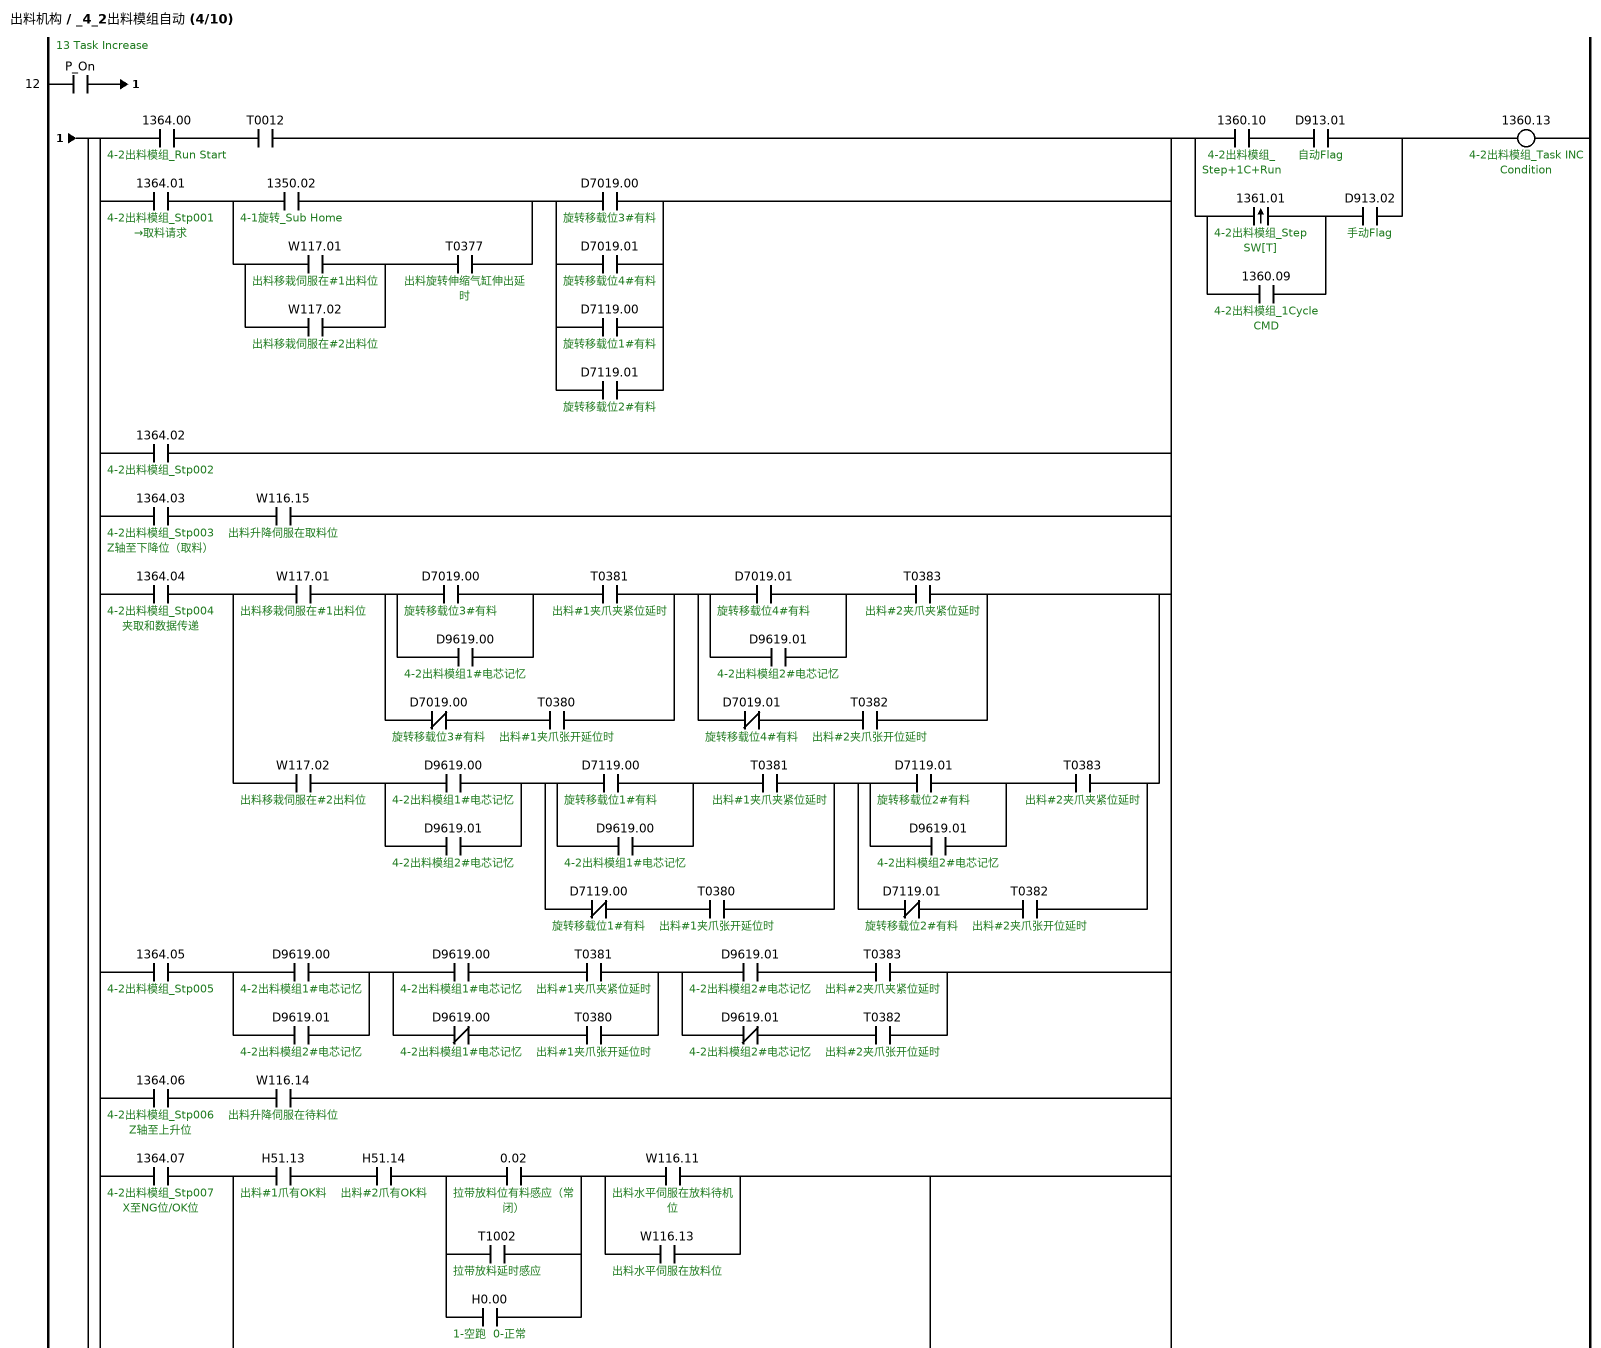
; [picture p384: 出料机构 / _4_2出料模组自动, rungs 12-12]

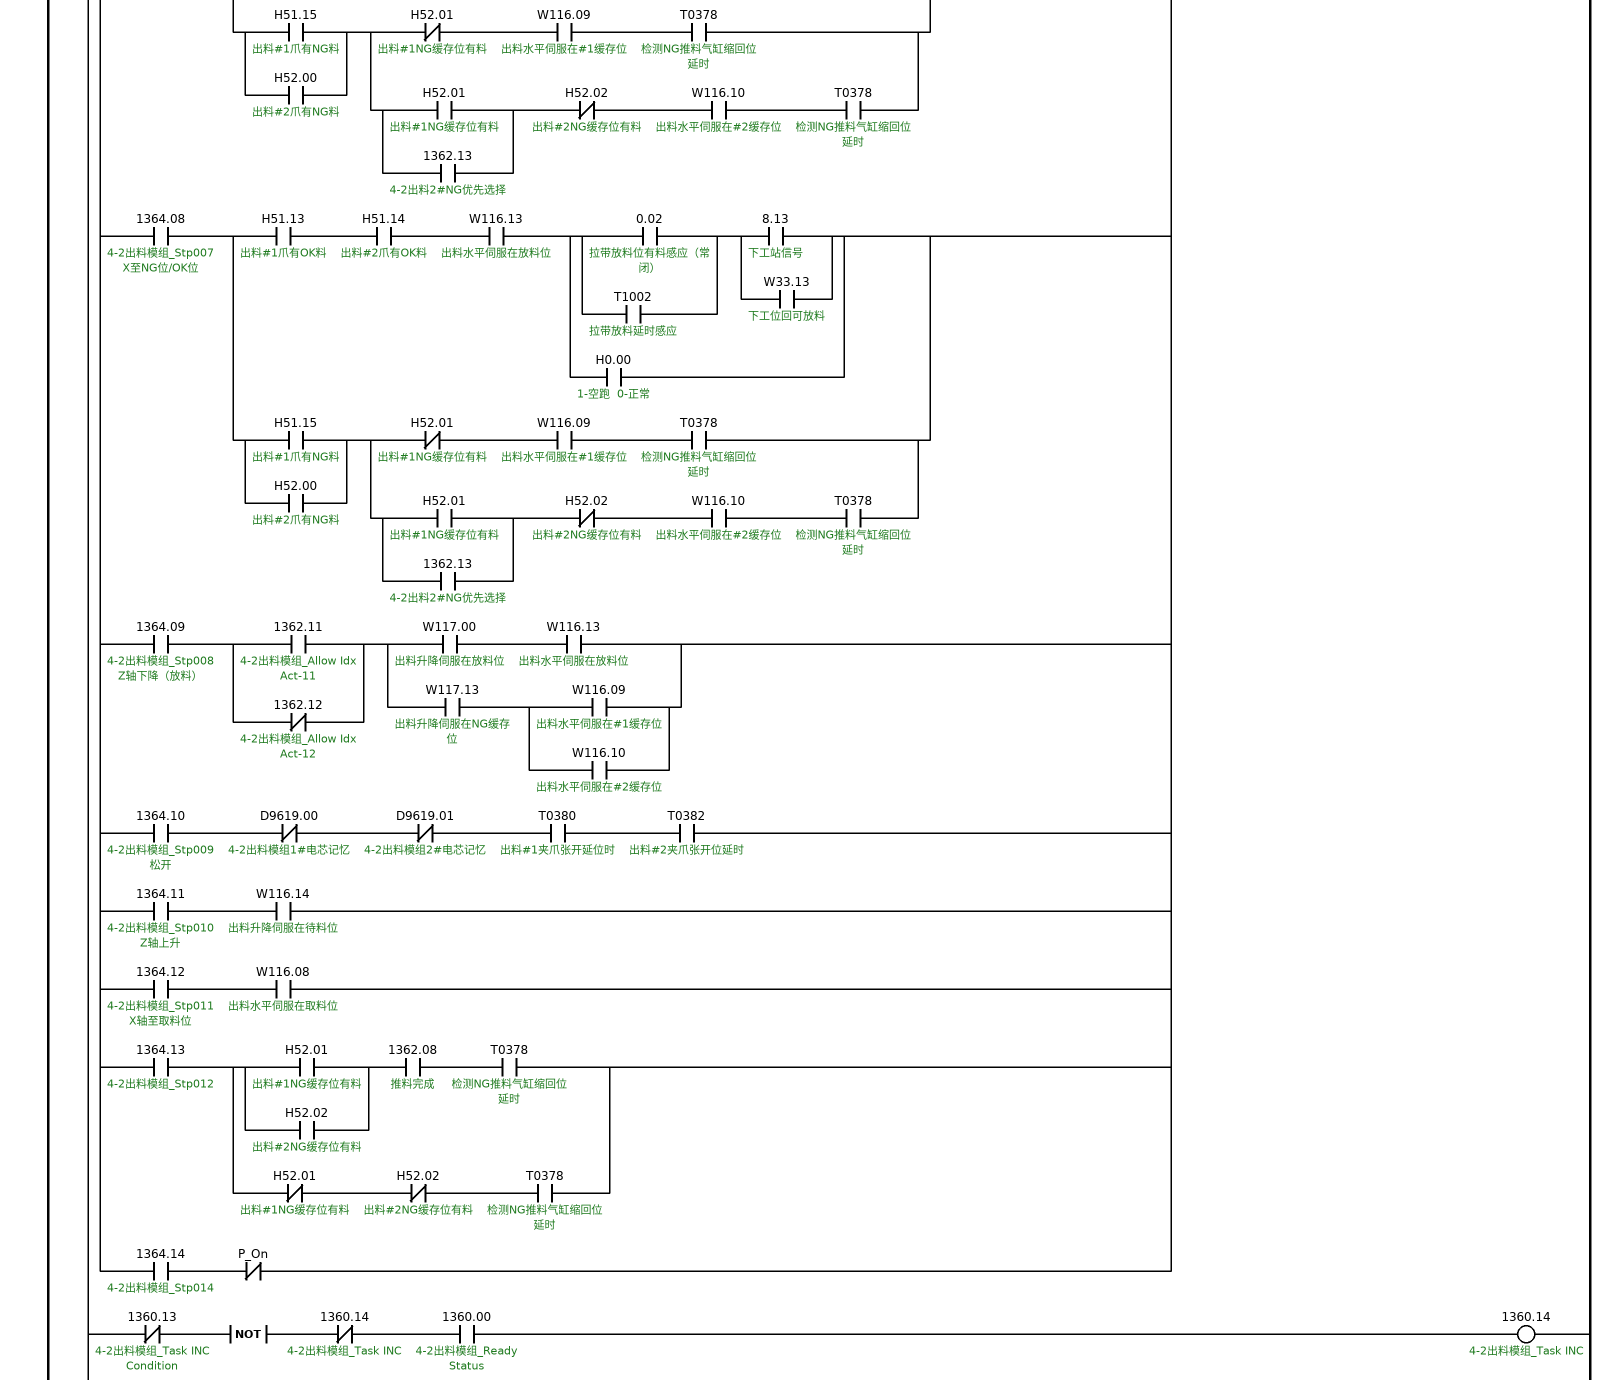

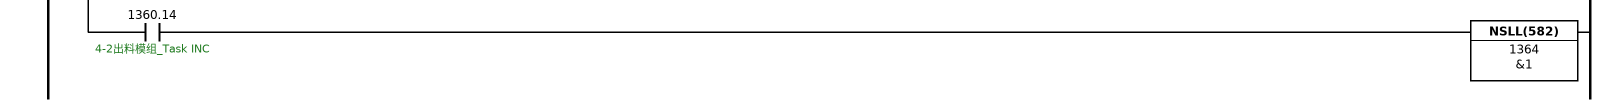
; rung 12: 13 Task Increase
LD P_On
OUT TR0
LD 1364.00  ; 4-2出料模组_Run Start
AND T0012
LD 1364.01  ; 4-2出料模组_Stp001 →取料请求
LD 1350.02  ; 4-1旋转_Sub Home
LD W117.01  ; 出料移栽伺服在#1出料位
OR W117.02  ; 出料移栽伺服在#2出料位
AND T0377  ; 出料旋转伸缩气缸伸出延时
ORLD
ANDLD
LD D7019.00  ; 旋转移载位3#有料
OR D7019.01  ; 旋转移载位4#有料
OR D7119.00  ; 旋转移载位1#有料
OR D7119.01  ; 旋转移载位2#有料
ANDLD
ORLD
OR 1364.02  ; 4-2出料模组_Stp002
LD 1364.03  ; 4-2出料模组_Stp003 Z轴至下降位（取料）
AND W116.15  ; 出料升降伺服在取料位
ORLD
LD 1364.04  ; 4-2出料模组_Stp004 夹取和数据传递
LD W117.01  ; 出料移栽伺服在#1出料位
LD D7019.00  ; 旋转移载位3#有料
OR D9619.00  ; 4-2出料模组1#电芯记忆
AND T0381  ; 出料#1夹爪夹紧位延时
LDNOT D7019.00  ; 旋转移载位3#有料
AND T0380  ; 出料#1夹爪张开延位时
ORLD
ANDLD
LD D7019.01  ; 旋转移载位4#有料
OR D9619.01  ; 4-2出料模组2#电芯记忆
AND T0383  ; 出料#2夹爪夹紧位延时
LDNOT D7019.01  ; 旋转移载位4#有料
AND T0382  ; 出料#2夹爪张开位延时
ORLD
ANDLD
LD W117.02  ; 出料移栽伺服在#2出料位
LD D9619.00  ; 4-2出料模组1#电芯记忆
OR D9619.01  ; 4-2出料模组2#电芯记忆
ANDLD
LD D7119.00  ; 旋转移载位1#有料
OR D9619.00  ; 4-2出料模组1#电芯记忆
AND T0381  ; 出料#1夹爪夹紧位延时
LDNOT D7119.00  ; 旋转移载位1#有料
AND T0380  ; 出料#1夹爪张开延位时
ORLD
ANDLD
LD D7119.01  ; 旋转移载位2#有料
OR D9619.01  ; 4-2出料模组2#电芯记忆
AND T0383  ; 出料#2夹爪夹紧位延时
LDNOT D7119.01  ; 旋转移载位2#有料
AND T0382  ; 出料#2夹爪张开位延时
ORLD
ANDLD
ORLD
ANDLD
ORLD
LD 1364.05  ; 4-2出料模组_Stp005
LD D9619.00  ; 4-2出料模组1#电芯记忆
OR D9619.01  ; 4-2出料模组2#电芯记忆
ANDLD
LD D9619.00  ; 4-2出料模组1#电芯记忆
AND T0381  ; 出料#1夹爪夹紧位延时
LDNOT D9619.00  ; 4-2出料模组1#电芯记忆
AND T0380  ; 出料#1夹爪张开延位时
ORLD
ANDLD
LD D9619.01  ; 4-2出料模组2#电芯记忆
AND T0383  ; 出料#2夹爪夹紧位延时
LDNOT D9619.01  ; 4-2出料模组2#电芯记忆
AND T0382  ; 出料#2夹爪张开位延时
ORLD
ANDLD
ORLD
LD 1364.06  ; 4-2出料模组_Stp006 Z轴至上升位
AND W116.14  ; 出料升降伺服在待料位
ORLD
LD 1364.07  ; 4-2出料模组_Stp007 X至NG位/OK位
LD H51.13  ; 出料#1爪有OK料
AND H51.14  ; 出料#2爪有OK料
LD 0.02  ; 拉带放料位有料感应（常闭）
OR T1002  ; 拉带放料延时感应
OR H0.00  ; 1-空跑  0-正常
ANDLD
LD W116.11  ; 出料水平伺服在放料待机位
OR W116.13  ; 出料水平伺服在放料位
ANDLD
LD H51.15  ; 出料#1爪有NG料
OR H52.00  ; 出料#2爪有NG料
LDNOT H52.01  ; 出料#1NG缓存位有料
AND W116.09  ; 出料水平伺服在#1缓存位
AND T0378  ; 检测NG推料气缸缩回位延时
LD H52.01  ; 出料#1NG缓存位有料
OR 1362.13  ; 4-2出料2#NG优先选择
ANDNOT H52.02  ; 出料#2NG缓存位有料
AND W116.10  ; 出料水平伺服在#2缓存位
AND T0378  ; 检测NG推料气缸缩回位延时
ORLD
ANDLD
ORLD
ANDLD
ORLD
LD 1364.08  ; 4-2出料模组_Stp007 X至NG位/OK位
LD H51.13  ; 出料#1爪有OK料
AND H51.14  ; 出料#2爪有OK料
AND W116.13  ; 出料水平伺服在放料位
LD 0.02  ; 拉带放料位有料感应（常闭）
OR T1002  ; 拉带放料延时感应
LD 8.13  ; 下工站信号
OR W33.13  ; 下工位回可放料
ANDLD
OR H0.00  ; 1-空跑  0-正常
ANDLD
LD H51.15  ; 出料#1爪有NG料
OR H52.00  ; 出料#2爪有NG料
LDNOT H52.01  ; 出料#1NG缓存位有料
AND W116.09  ; 出料水平伺服在#1缓存位
AND T0378  ; 检测NG推料气缸缩回位延时
LD H52.01  ; 出料#1NG缓存位有料
OR 1362.13  ; 4-2出料2#NG优先选择
ANDNOT H52.02  ; 出料#2NG缓存位有料
AND W116.10  ; 出料水平伺服在#2缓存位
AND T0378  ; 检测NG推料气缸缩回位延时
ORLD
ANDLD
ORLD
ANDLD
ORLD
LD 1364.09  ; 4-2出料模组_Stp008 Z轴下降（放料）
LD 1362.11  ; 4-2出料模组_Allow Idx Act-11
ORNOT 1362.12  ; 4-2出料模组_Allow Idx Act-12
ANDLD
LD W117.00  ; 出料升降伺服在放料位
AND W116.13  ; 出料水平伺服在放料位
LD W117.13  ; 出料升降伺服在NG缓存位
LD W116.09  ; 出料水平伺服在#1缓存位
OR W116.10  ; 出料水平伺服在#2缓存位
ANDLD
ORLD
ANDLD
ORLD
LD 1364.10  ; 4-2出料模组_Stp009 松开
ANDNOT D9619.00  ; 4-2出料模组1#电芯记忆
ANDNOT D9619.01  ; 4-2出料模组2#电芯记忆
AND T0380  ; 出料#1夹爪张开延位时
AND T0382  ; 出料#2夹爪张开位延时
ORLD
LD 1364.11  ; 4-2出料模组_Stp010 Z轴上升
AND W116.14  ; 出料升降伺服在待料位
ORLD
LD 1364.12  ; 4-2出料模组_Stp011 X轴至取料位
AND W116.08  ; 出料水平伺服在取料位
ORLD
LD 1364.13  ; 4-2出料模组_Stp012
LD H52.01  ; 出料#1NG缓存位有料
OR H52.02  ; 出料#2NG缓存位有料
AND 1362.08  ; 推料完成
AND T0378  ; 检测NG推料气缸缩回位延时
LDNOT H52.01  ; 出料#1NG缓存位有料
ANDNOT H52.02  ; 出料#2NG缓存位有料
AND T0378  ; 检测NG推料气缸缩回位延时
ORLD
ANDLD
ORLD
LD 1364.14  ; 4-2出料模组_Stp014
ANDNOT P_On
ORLD
ANDLD
LD 1360.10  ; 4-2出料模组_Step+1C+Run
AND D913.01  ; 自动Flag
@LD 1361.01  ; 4-2出料模组_Step SW[T]
OR 1360.09  ; 4-2出料模组_1Cycle CMD
AND D913.02  ; 手动Flag
ORLD
ANDLD
OUT 1360.13  ; 4-2出料模组_Task INC Condition
LD TR0
ANDNOT 1360.13  ; 4-2出料模组_Task INC Condition
NOT(520)
ANDNOT 1360.14  ; 4-2出料模组_Task INC
AND 1360.00  ; 4-2出料模组_Ready Status
OUT 1360.14  ; 4-2出料模组_Task INC
LD TR0
AND 1360.14  ; 4-2出料模组_Task INC
NSLL(582) 1364 &1

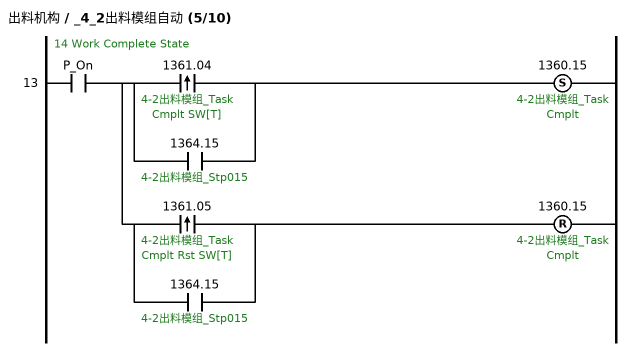
; rung 13: 14 Work Complete State
LD P_On
OUT TR0
@LD 1361.04  ; 4-2出料模组_Task Cmplt SW[T]
OR 1364.15  ; 4-2出料模组_Stp015
ANDLD
SET 1360.15  ; 4-2出料模组_Task Cmplt
LD TR0
@LD 1361.05  ; 4-2出料模组_Task Cmplt Rst SW[T]
OR 1364.15  ; 4-2出料模组_Stp015
ANDLD
RSET 1360.15  ; 4-2出料模组_Task Cmplt

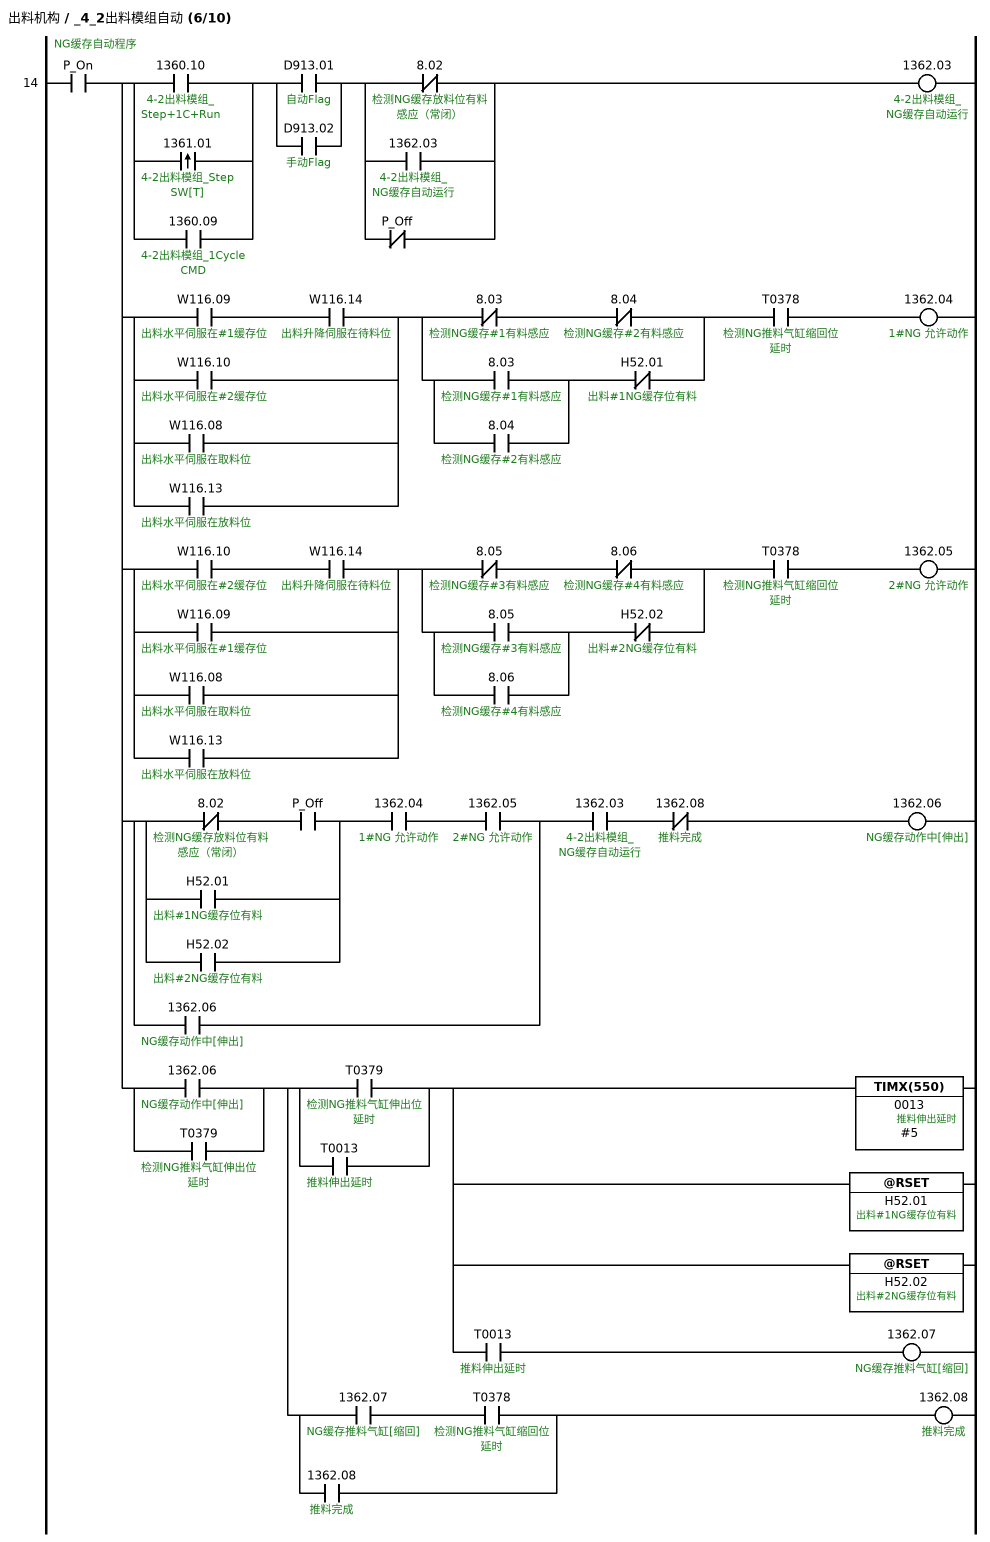
; rung 14: NG缓存自动程序
LD P_On
OUT TR0
LD 1360.10  ; 4-2出料模组_Step+1C+Run
@OR 1361.01  ; 4-2出料模组_Step SW[T]
OR 1360.09  ; 4-2出料模组_1Cycle CMD
ANDLD
LD D913.01  ; 自动Flag
OR D913.02  ; 手动Flag
ANDLD
LDNOT 8.02  ; 检测NG缓存放料位有料感应（常闭）
OR 1362.03  ; 4-2出料模组_NG缓存自动运行
ORNOT P_Off
ANDLD
OUT 1362.03  ; 4-2出料模组_NG缓存自动运行
LD TR0
LD W116.09  ; 出料水平伺服在#1缓存位
AND W116.14  ; 出料升降伺服在待料位
OR W116.10  ; 出料水平伺服在#2缓存位
OR W116.08  ; 出料水平伺服在取料位
OR W116.13  ; 出料水平伺服在放料位
ANDLD
LDNOT 8.03  ; 检测NG缓存#1有料感应
ANDNOT 8.04  ; 检测NG缓存#2有料感应
LD 8.03  ; 检测NG缓存#1有料感应
OR 8.04  ; 检测NG缓存#2有料感应
ANDNOT H52.01  ; 出料#1NG缓存位有料
ORLD
ANDLD
AND T0378  ; 检测NG推料气缸缩回位延时
OUT 1362.04  ; 1#NG 允许动作
LD TR0
LD W116.10  ; 出料水平伺服在#2缓存位
AND W116.14  ; 出料升降伺服在待料位
OR W116.09  ; 出料水平伺服在#1缓存位
OR W116.08  ; 出料水平伺服在取料位
OR W116.13  ; 出料水平伺服在放料位
ANDLD
LDNOT 8.05  ; 检测NG缓存#3有料感应
ANDNOT 8.06  ; 检测NG缓存#4有料感应
LD 8.05  ; 检测NG缓存#3有料感应
OR 8.06  ; 检测NG缓存#4有料感应
ANDNOT H52.02  ; 出料#2NG缓存位有料
ORLD
ANDLD
AND T0378  ; 检测NG推料气缸缩回位延时
OUT 1362.05  ; 2#NG 允许动作
LD TR0
LDNOT 8.02  ; 检测NG缓存放料位有料感应（常闭）
AND P_Off
OR H52.01  ; 出料#1NG缓存位有料
OR H52.02  ; 出料#2NG缓存位有料
AND 1362.04  ; 1#NG 允许动作
AND 1362.05  ; 2#NG 允许动作
OR 1362.06  ; NG缓存动作中[伸出]
ANDLD
AND 1362.03  ; 4-2出料模组_NG缓存自动运行
ANDNOT 1362.08  ; 推料完成
OUT 1362.06  ; NG缓存动作中[伸出]
LD TR0
LD 1362.06  ; NG缓存动作中[伸出]
OR T0379  ; 检测NG推料气缸伸出位延时
ANDLD
OUT TR0
LD T0379  ; 检测NG推料气缸伸出位延时
OR T0013  ; 推料伸出延时
ANDLD
TIMX(550) 0013 #5  ; 推料伸出延时
@RSET H52.01  ; 出料#1NG缓存位有料
@RSET H52.02  ; 出料#2NG缓存位有料
AND T0013  ; 推料伸出延时
OUT 1362.07  ; NG缓存推料气缸[缩回]
LD TR0
LD 1362.07  ; NG缓存推料气缸[缩回]
AND T0378  ; 检测NG推料气缸缩回位延时
OR 1362.08  ; 推料完成
ANDLD
OUT 1362.08  ; 推料完成

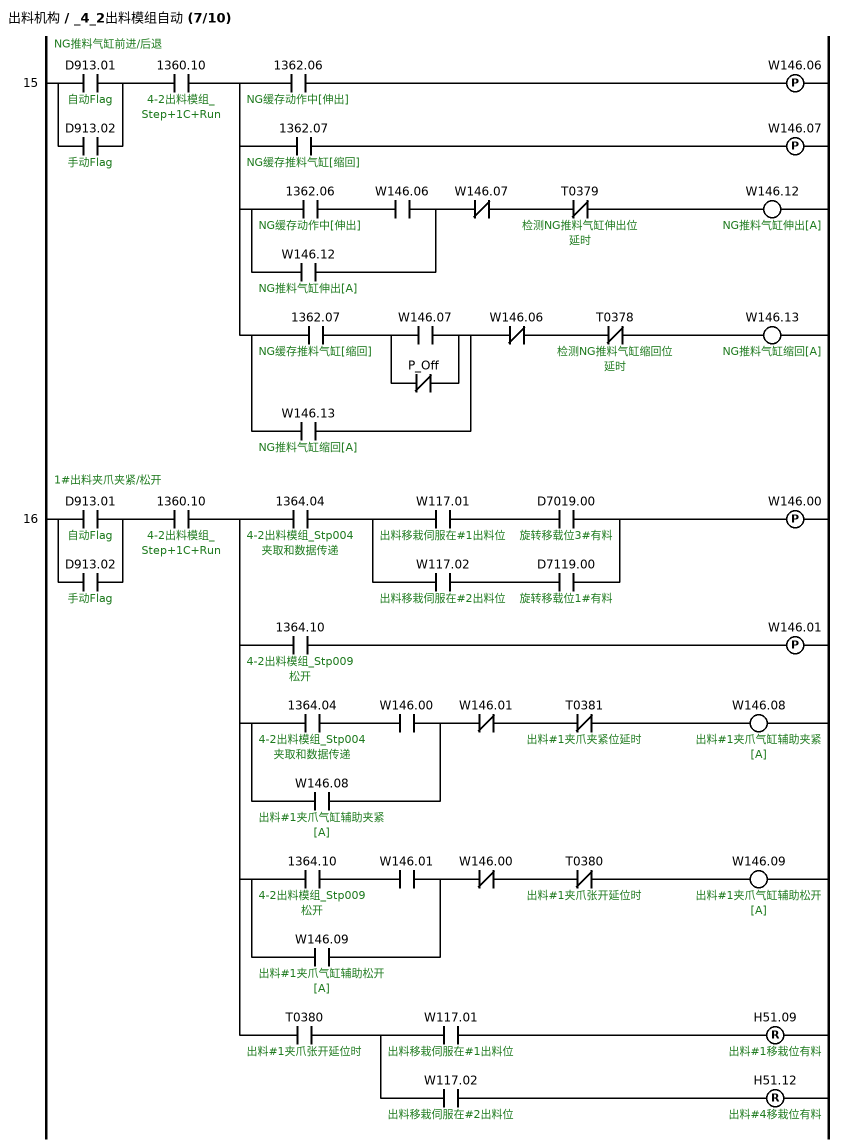
; rung 15: NG推料气缸前进/后退
LD D913.01  ; 自动Flag
OR D913.02  ; 手动Flag
AND 1360.10  ; 4-2出料模组_Step+1C+Run
OUT TR0
AND 1362.06  ; NG缓存动作中[伸出]
DIFU(013) W146.06
LD TR0
AND 1362.07  ; NG缓存推料气缸[缩回]
DIFU(013) W146.07
LD TR0
LD 1362.06  ; NG缓存动作中[伸出]
AND W146.06
OR W146.12  ; NG推料气缸伸出[A]
ANDLD
ANDNOT W146.07
ANDNOT T0379  ; 检测NG推料气缸伸出位延时
OUT W146.12  ; NG推料气缸伸出[A]
LD TR0
LD 1362.07  ; NG缓存推料气缸[缩回]
LD W146.07
ORNOT P_Off
ANDLD
OR W146.13  ; NG推料气缸缩回[A]
ANDLD
ANDNOT W146.06
ANDNOT T0378  ; 检测NG推料气缸缩回位延时
OUT W146.13  ; NG推料气缸缩回[A]
; rung 16: 1#出料夹爪夹紧/松开
LD D913.01  ; 自动Flag
OR D913.02  ; 手动Flag
AND 1360.10  ; 4-2出料模组_Step+1C+Run
OUT TR0
AND 1364.04  ; 4-2出料模组_Stp004 夹取和数据传递
LD W117.01  ; 出料移栽伺服在#1出料位
AND D7019.00  ; 旋转移载位3#有料
LD W117.02  ; 出料移栽伺服在#2出料位
AND D7119.00  ; 旋转移载位1#有料
ORLD
ANDLD
DIFU(013) W146.00
LD TR0
AND 1364.10  ; 4-2出料模组_Stp009 松开
DIFU(013) W146.01
LD TR0
LD 1364.04  ; 4-2出料模组_Stp004 夹取和数据传递
AND W146.00
OR W146.08  ; 出料#1夹爪气缸辅助夹紧[A]
ANDLD
ANDNOT W146.01
ANDNOT T0381  ; 出料#1夹爪夹紧位延时
OUT W146.08  ; 出料#1夹爪气缸辅助夹紧[A]
LD TR0
LD 1364.10  ; 4-2出料模组_Stp009 松开
AND W146.01
OR W146.09  ; 出料#1夹爪气缸辅助松开[A]
ANDLD
ANDNOT W146.00
ANDNOT T0380  ; 出料#1夹爪张开延位时
OUT W146.09  ; 出料#1夹爪气缸辅助松开[A]
LD TR0
AND T0380  ; 出料#1夹爪张开延位时
OUT TR0
AND W117.01  ; 出料移栽伺服在#1出料位
RSET H51.09  ; 出料#1移栽位有料
LD TR0
AND W117.02  ; 出料移栽伺服在#2出料位
RSET H51.12  ; 出料#4移栽位有料

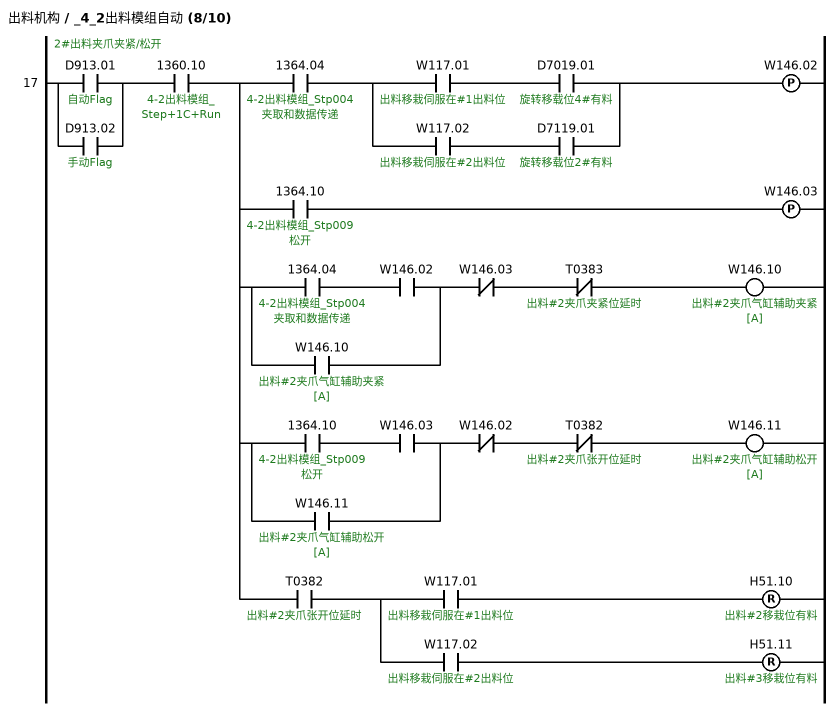
; rung 17: 2#出料夹爪夹紧/松开
LD D913.01  ; 自动Flag
OR D913.02  ; 手动Flag
AND 1360.10  ; 4-2出料模组_Step+1C+Run
OUT TR0
AND 1364.04  ; 4-2出料模组_Stp004 夹取和数据传递
LD W117.01  ; 出料移栽伺服在#1出料位
AND D7019.01  ; 旋转移载位4#有料
LD W117.02  ; 出料移栽伺服在#2出料位
AND D7119.01  ; 旋转移载位2#有料
ORLD
ANDLD
DIFU(013) W146.02
LD TR0
AND 1364.10  ; 4-2出料模组_Stp009 松开
DIFU(013) W146.03
LD TR0
LD 1364.04  ; 4-2出料模组_Stp004 夹取和数据传递
AND W146.02
OR W146.10  ; 出料#2夹爪气缸辅助夹紧[A]
ANDLD
ANDNOT W146.03
ANDNOT T0383  ; 出料#2夹爪夹紧位延时
OUT W146.10  ; 出料#2夹爪气缸辅助夹紧[A]
LD TR0
LD 1364.10  ; 4-2出料模组_Stp009 松开
AND W146.03
OR W146.11  ; 出料#2夹爪气缸辅助松开[A]
ANDLD
ANDNOT W146.02
ANDNOT T0382  ; 出料#2夹爪张开位延时
OUT W146.11  ; 出料#2夹爪气缸辅助松开[A]
LD TR0
AND T0382  ; 出料#2夹爪张开位延时
OUT TR0
AND W117.01  ; 出料移栽伺服在#1出料位
RSET H51.10  ; 出料#2移栽位有料
LD TR0
AND W117.02  ; 出料移栽伺服在#2出料位
RSET H51.11  ; 出料#3移栽位有料

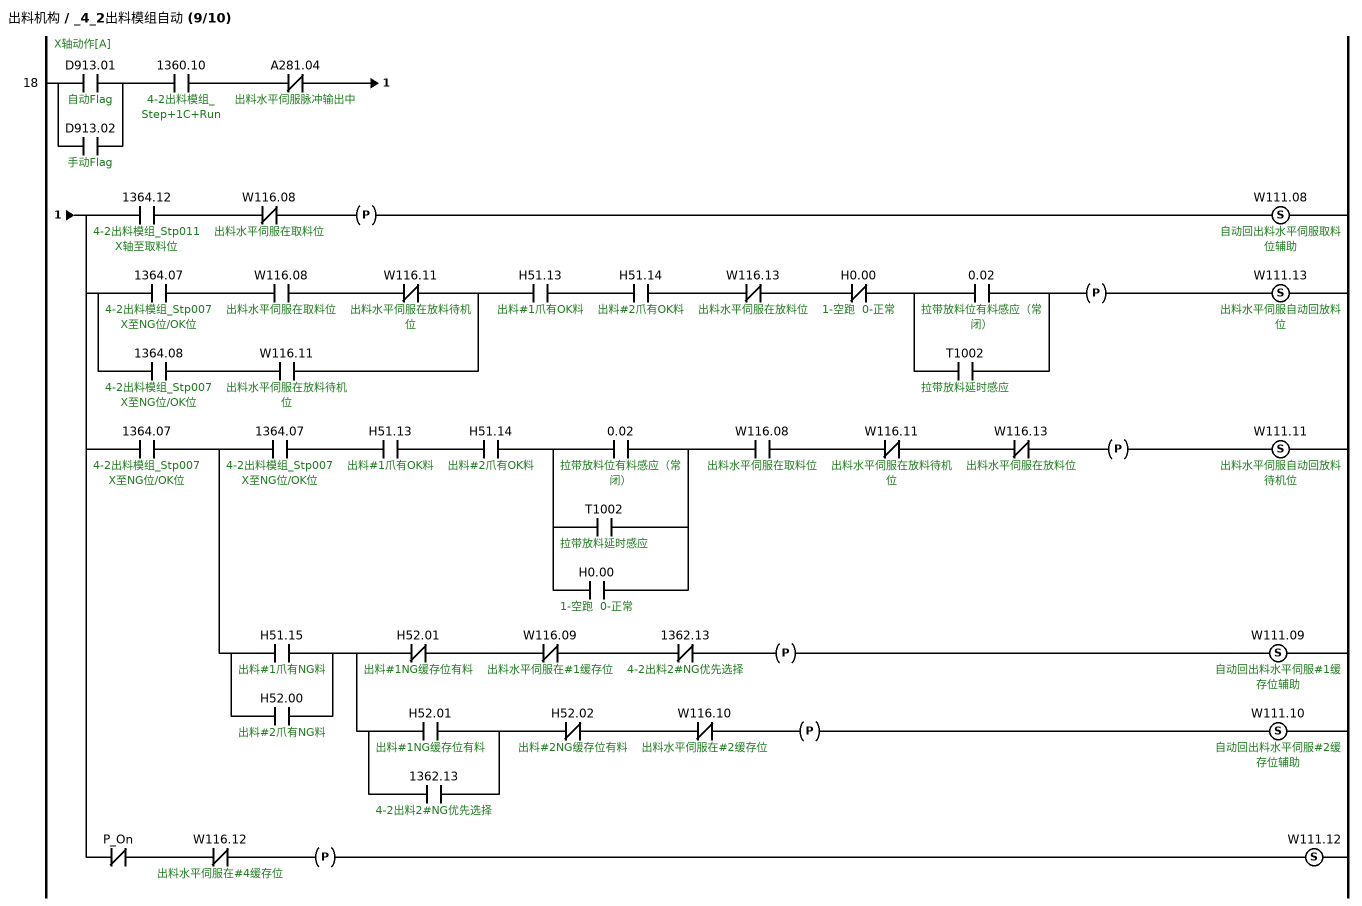
; rung 18: X轴动作[A]
LD D913.01  ; 自动Flag
OR D913.02  ; 手动Flag
AND 1360.10  ; 4-2出料模组_Step+1C+Run
ANDNOT A281.04  ; 出料水平伺服脉冲输出中
OUT TR0
AND 1364.12  ; 4-2出料模组_Stp011 X轴至取料位
ANDNOT W116.08  ; 出料水平伺服在取料位
UP(521)
SET W111.08  ; 自动回出料水平伺服取料位辅助
LD TR0
LD 1364.07  ; 4-2出料模组_Stp007 X至NG位/OK位
AND W116.08  ; 出料水平伺服在取料位
ANDNOT W116.11  ; 出料水平伺服在放料待机位
LD 1364.08  ; 4-2出料模组_Stp007 X至NG位/OK位
AND W116.11  ; 出料水平伺服在放料待机位
ORLD
ANDLD
AND H51.13  ; 出料#1爪有OK料
AND H51.14  ; 出料#2爪有OK料
ANDNOT W116.13  ; 出料水平伺服在放料位
ANDNOT H0.00  ; 1-空跑  0-正常
LD 0.02  ; 拉带放料位有料感应（常闭）
OR T1002  ; 拉带放料延时感应
ANDLD
UP(521)
SET W111.13  ; 出料水平伺服自动回放料位
LD TR0
AND 1364.07  ; 4-2出料模组_Stp007 X至NG位/OK位
OUT TR1
AND 1364.07  ; 4-2出料模组_Stp007 X至NG位/OK位
AND H51.13  ; 出料#1爪有OK料
AND H51.14  ; 出料#2爪有OK料
LD 0.02  ; 拉带放料位有料感应（常闭）
OR T1002  ; 拉带放料延时感应
OR H0.00  ; 1-空跑  0-正常
ANDLD
AND W116.08  ; 出料水平伺服在取料位
ANDNOT W116.11  ; 出料水平伺服在放料待机位
ANDNOT W116.13  ; 出料水平伺服在放料位
UP(521)
SET W111.11  ; 出料水平伺服自动回放料待机位
LD TR1
LD H51.15  ; 出料#1爪有NG料
OR H52.00  ; 出料#2爪有NG料
ANDLD
OUT TR1
ANDNOT H52.01  ; 出料#1NG缓存位有料
ANDNOT W116.09  ; 出料水平伺服在#1缓存位
ANDNOT 1362.13  ; 4-2出料2#NG优先选择
UP(521)
SET W111.09  ; 自动回出料水平伺服#1缓存位辅助
LD TR1
LD H52.01  ; 出料#1NG缓存位有料
OR 1362.13  ; 4-2出料2#NG优先选择
ANDLD
ANDNOT H52.02  ; 出料#2NG缓存位有料
ANDNOT W116.10  ; 出料水平伺服在#2缓存位
UP(521)
SET W111.10  ; 自动回出料水平伺服#2缓存位辅助
LD TR0
ANDNOT P_On
ANDNOT W116.12  ; 出料水平伺服在#4缓存位
UP(521)
SET W111.12

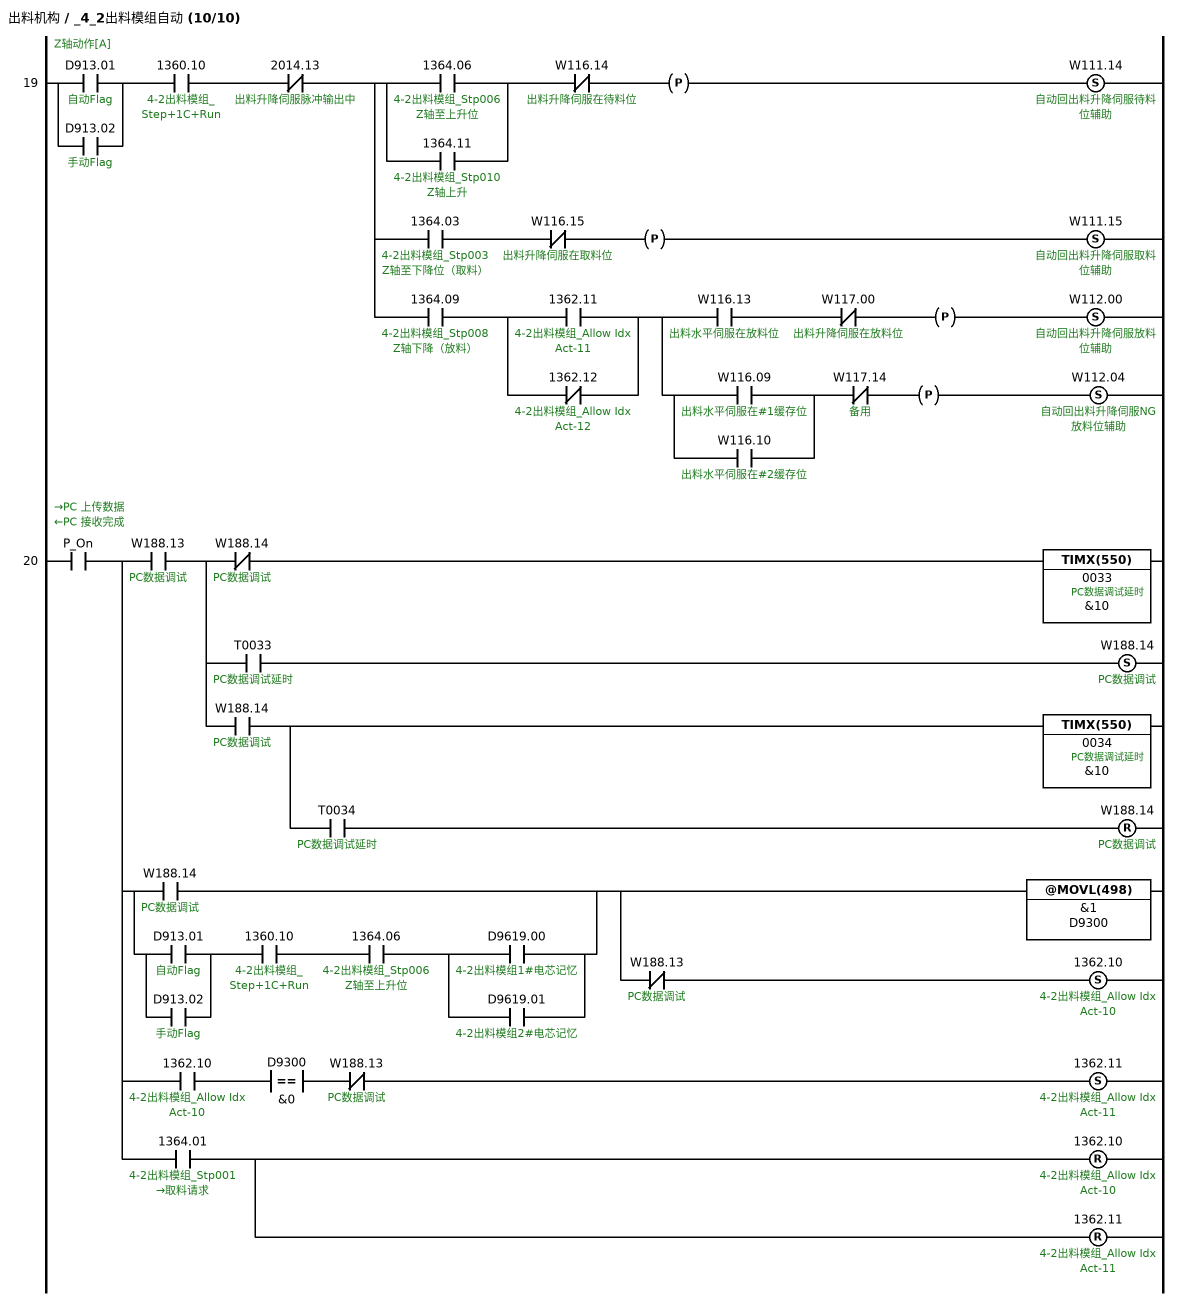
; rung 19: Z轴动作[A]
LD D913.01  ; 自动Flag
OR D913.02  ; 手动Flag
AND 1360.10  ; 4-2出料模组_Step+1C+Run
ANDNOT 2014.13  ; 出料升降伺服脉冲输出中
OUT TR0
LD 1364.06  ; 4-2出料模组_Stp006 Z轴至上升位
OR 1364.11  ; 4-2出料模组_Stp010 Z轴上升
ANDLD
ANDNOT W116.14  ; 出料升降伺服在待料位
UP(521)
SET W111.14  ; 自动回出料升降伺服待料位辅助
LD TR0
AND 1364.03  ; 4-2出料模组_Stp003 Z轴至下降位（取料）
ANDNOT W116.15  ; 出料升降伺服在取料位
UP(521)
SET W111.15  ; 自动回出料升降伺服取料位辅助
LD TR0
AND 1364.09  ; 4-2出料模组_Stp008 Z轴下降（放料）
LD 1362.11  ; 4-2出料模组_Allow Idx Act-11
ORNOT 1362.12  ; 4-2出料模组_Allow Idx Act-12
ANDLD
OUT TR0
AND W116.13  ; 出料水平伺服在放料位
ANDNOT W117.00  ; 出料升降伺服在放料位
UP(521)
SET W112.00  ; 自动回出料升降伺服放料位辅助
LD TR0
LD W116.09  ; 出料水平伺服在#1缓存位
OR W116.10  ; 出料水平伺服在#2缓存位
ANDLD
ANDNOT W117.14  ; 备用
UP(521)
SET W112.04  ; 自动回出料升降伺服NG放料位辅助
; rung 20: →PC 上传数据 / ←PC 接收完成
LD P_On
OUT TR0
AND W188.13  ; PC数据调试
OUT TR1
ANDNOT W188.14  ; PC数据调试
TIMX(550) 0033 &10  ; PC数据调试延时
LD TR1
AND T0033  ; PC数据调试延时
SET W188.14  ; PC数据调试
LD TR1
AND W188.14  ; PC数据调试
TIMX(550) 0034 &10  ; PC数据调试延时
AND T0034  ; PC数据调试延时
RSET W188.14  ; PC数据调试
LD TR0
LD W188.14  ; PC数据调试
LD D913.01  ; 自动Flag
OR D913.02  ; 手动Flag
AND 1360.10  ; 4-2出料模组_Step+1C+Run
AND 1364.06  ; 4-2出料模组_Stp006 Z轴至上升位
LD D9619.00  ; 4-2出料模组1#电芯记忆
OR D9619.01  ; 4-2出料模组2#电芯记忆
ANDLD
ORLD
ANDLD
@MOVL(498) &1 D9300
ANDNOT W188.13  ; PC数据调试
SET 1362.10  ; 4-2出料模组_Allow Idx Act-10
LD TR0
AND 1362.10  ; 4-2出料模组_Allow Idx Act-10
AND=SL(303) D9300 &0
ANDNOT W188.13  ; PC数据调试
SET 1362.11  ; 4-2出料模组_Allow Idx Act-11
LD TR0
AND 1364.01  ; 4-2出料模组_Stp001 →取料请求
RSET 1362.10  ; 4-2出料模组_Allow Idx Act-10
RSET 1362.11  ; 4-2出料模组_Allow Idx Act-11

### Section 初始化

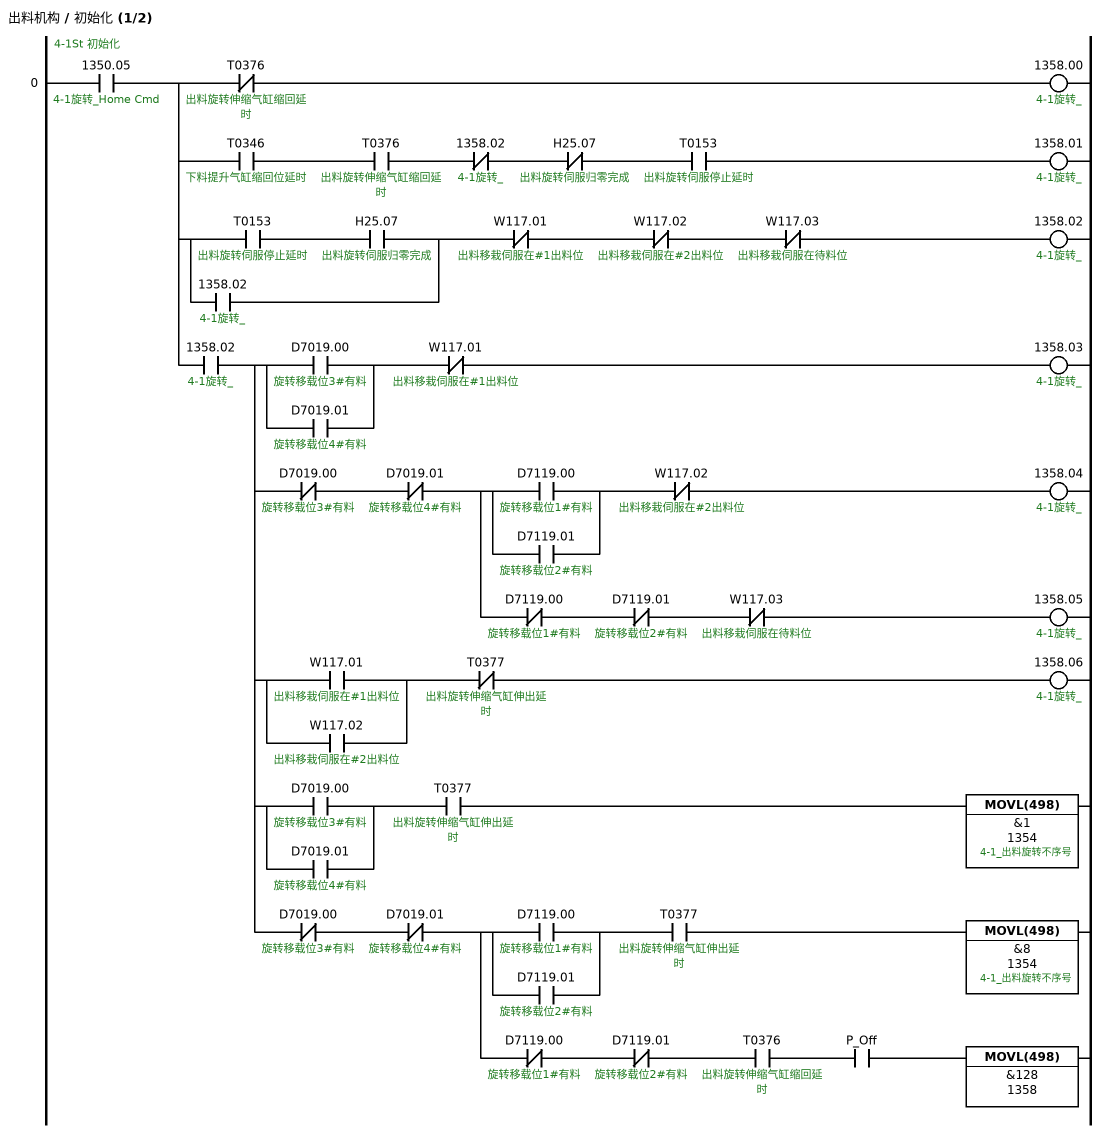
; rung 0: 4-1St 初始化
LD 1350.05  ; 4-1旋转_Home Cmd
OUT TR0
ANDNOT T0376  ; 出料旋转伸缩气缸缩回延时
OUT 1358.00  ; 4-1旋转_
LD TR0
AND T0346  ; 下料提升气缸缩回位延时
AND T0376  ; 出料旋转伸缩气缸缩回延时
ANDNOT 1358.02  ; 4-1旋转_
ANDNOT H25.07  ; 出料旋转伺服归零完成
AND T0153  ; 出料旋转伺服停止延时
OUT 1358.01  ; 4-1旋转_
LD TR0
LD T0153  ; 出料旋转伺服停止延时
AND H25.07  ; 出料旋转伺服归零完成
OR 1358.02  ; 4-1旋转_
ANDLD
ANDNOT W117.01  ; 出料移栽伺服在#1出料位
ANDNOT W117.02  ; 出料移栽伺服在#2出料位
ANDNOT W117.03  ; 出料移栽伺服在待料位
OUT 1358.02  ; 4-1旋转_
LD TR0
AND 1358.02  ; 4-1旋转_
OUT TR0
LD D7019.00  ; 旋转移载位3#有料
OR D7019.01  ; 旋转移载位4#有料
ANDLD
ANDNOT W117.01  ; 出料移栽伺服在#1出料位
OUT 1358.03  ; 4-1旋转_
LD TR0
ANDNOT D7019.00  ; 旋转移载位3#有料
ANDNOT D7019.01  ; 旋转移载位4#有料
OUT TR1
LD D7119.00  ; 旋转移载位1#有料
OR D7119.01  ; 旋转移载位2#有料
ANDLD
ANDNOT W117.02  ; 出料移栽伺服在#2出料位
OUT 1358.04  ; 4-1旋转_
LD TR1
ANDNOT D7119.00  ; 旋转移载位1#有料
ANDNOT D7119.01  ; 旋转移载位2#有料
ANDNOT W117.03  ; 出料移栽伺服在待料位
OUT 1358.05  ; 4-1旋转_
LD TR0
LD W117.01  ; 出料移栽伺服在#1出料位
OR W117.02  ; 出料移栽伺服在#2出料位
ANDLD
ANDNOT T0377  ; 出料旋转伸缩气缸伸出延时
OUT 1358.06  ; 4-1旋转_
LD TR0
LD D7019.00  ; 旋转移载位3#有料
OR D7019.01  ; 旋转移载位4#有料
ANDLD
AND T0377  ; 出料旋转伸缩气缸伸出延时
MOVL(498) &1 1354  ; 4-1_出料旋转不序号
LD TR0
ANDNOT D7019.00  ; 旋转移载位3#有料
ANDNOT D7019.01  ; 旋转移载位4#有料
OUT TR0
LD D7119.00  ; 旋转移载位1#有料
OR D7119.01  ; 旋转移载位2#有料
ANDLD
AND T0377  ; 出料旋转伸缩气缸伸出延时
MOVL(498) &8 1354  ; 4-1_出料旋转不序号
LD TR0
ANDNOT D7119.00  ; 旋转移载位1#有料
ANDNOT D7119.01  ; 旋转移载位2#有料
AND T0376  ; 出料旋转伸缩气缸缩回延时
AND P_Off
MOVL(498) &128 1358

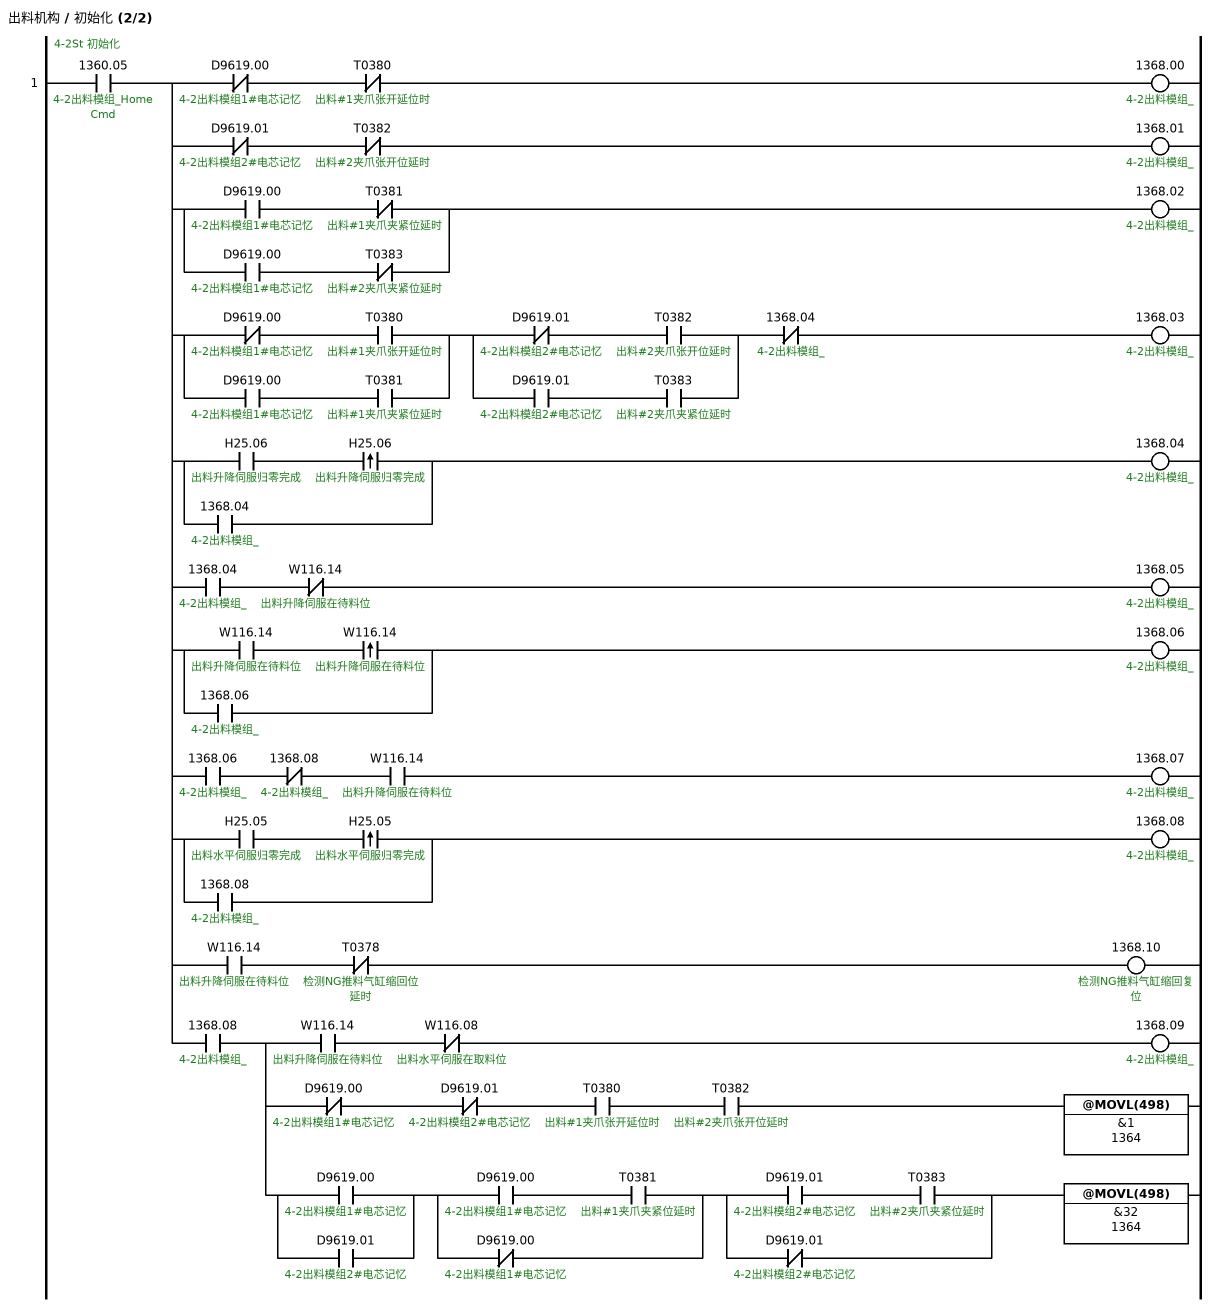
; rung 1: 4-2St 初始化
LD 1360.05  ; 4-2出料模组_Home Cmd
OUT TR0
ANDNOT D9619.00  ; 4-2出料模组1#电芯记忆
ANDNOT T0380  ; 出料#1夹爪张开延位时
OUT 1368.00  ; 4-2出料模组_
LD TR0
ANDNOT D9619.01  ; 4-2出料模组2#电芯记忆
ANDNOT T0382  ; 出料#2夹爪张开位延时
OUT 1368.01  ; 4-2出料模组_
LD TR0
LD D9619.00  ; 4-2出料模组1#电芯记忆
ANDNOT T0381  ; 出料#1夹爪夹紧位延时
LD D9619.00  ; 4-2出料模组1#电芯记忆
ANDNOT T0383  ; 出料#2夹爪夹紧位延时
ORLD
ANDLD
OUT 1368.02  ; 4-2出料模组_
LD TR0
LDNOT D9619.00  ; 4-2出料模组1#电芯记忆
AND T0380  ; 出料#1夹爪张开延位时
LD D9619.00  ; 4-2出料模组1#电芯记忆
AND T0381  ; 出料#1夹爪夹紧位延时
ORLD
ANDLD
LDNOT D9619.01  ; 4-2出料模组2#电芯记忆
AND T0382  ; 出料#2夹爪张开位延时
LD D9619.01  ; 4-2出料模组2#电芯记忆
AND T0383  ; 出料#2夹爪夹紧位延时
ORLD
ANDLD
ANDNOT 1368.04  ; 4-2出料模组_
OUT 1368.03  ; 4-2出料模组_
LD TR0
LD H25.06  ; 出料升降伺服归零完成
@AND H25.06  ; 出料升降伺服归零完成
OR 1368.04  ; 4-2出料模组_
ANDLD
OUT 1368.04  ; 4-2出料模组_
LD TR0
AND 1368.04  ; 4-2出料模组_
ANDNOT W116.14  ; 出料升降伺服在待料位
OUT 1368.05  ; 4-2出料模组_
LD TR0
LD W116.14  ; 出料升降伺服在待料位
@AND W116.14  ; 出料升降伺服在待料位
OR 1368.06  ; 4-2出料模组_
ANDLD
OUT 1368.06  ; 4-2出料模组_
LD TR0
AND 1368.06  ; 4-2出料模组_
ANDNOT 1368.08  ; 4-2出料模组_
AND W116.14  ; 出料升降伺服在待料位
OUT 1368.07  ; 4-2出料模组_
LD TR0
LD H25.05  ; 出料水平伺服归零完成
@AND H25.05  ; 出料水平伺服归零完成
OR 1368.08  ; 4-2出料模组_
ANDLD
OUT 1368.08  ; 4-2出料模组_
LD TR0
AND W116.14  ; 出料升降伺服在待料位
ANDNOT T0378  ; 检测NG推料气缸缩回位延时
OUT 1368.10  ; 检测NG推料气缸缩回复位
LD TR0
AND 1368.08  ; 4-2出料模组_
OUT TR0
AND W116.14  ; 出料升降伺服在待料位
ANDNOT W116.08  ; 出料水平伺服在取料位
OUT 1368.09  ; 4-2出料模组_
LD TR0
ANDNOT D9619.00  ; 4-2出料模组1#电芯记忆
ANDNOT D9619.01  ; 4-2出料模组2#电芯记忆
AND T0380  ; 出料#1夹爪张开延位时
AND T0382  ; 出料#2夹爪张开位延时
@MOVL(498) &1 1364
LD TR0
LD D9619.00  ; 4-2出料模组1#电芯记忆
OR D9619.01  ; 4-2出料模组2#电芯记忆
ANDLD
LD D9619.00  ; 4-2出料模组1#电芯记忆
AND T0381  ; 出料#1夹爪夹紧位延时
ORNOT D9619.00  ; 4-2出料模组1#电芯记忆
ANDLD
LD D9619.01  ; 4-2出料模组2#电芯记忆
AND T0383  ; 出料#2夹爪夹紧位延时
ORNOT D9619.01  ; 4-2出料模组2#电芯记忆
ANDLD
@MOVL(498) &32 1364

### Section END
; rung 0
END(001)